FUNCTION_BLOCK TestAwaitChainNormal
VAR
	nState: UDINT := 0;
	await: Await;

	fbClient: FB_IotHttpClient := (
		sHostName:='localhost',
		bKeepAlive:=TRUE,
		tConnectionTimeout:=T#10S,
		nHostPort:=8000
	);
	
	fbRequest: FB_IotHttpRequest;
	sEndpoint: STRING := '/hello-world';
	response: STRING(255);

	fbJson: FB_JsonDomParser;
	
	jsonDoc: SJsonValue;
	jsonMember: SJsonValue;
	isJsonMemberString: BOOL;
	
	RisingEdge: R_TRIG;
	
	bSend: BOOL;
	requestSent: BOOL;
	cycleCounter: INT := 0;
	lenResponse: INT := 0;
	
	// Awaitable Errors
	onRequestError: OnRequestError := (errorName:='Request error', onErrorStep:=500);
	onResponseError: OnRequestError := (errorName:='Response error', onErrorStep:=500);
	onJsonError: OnJsonError := (errorName:='Json error', onErrorStep:=500);
	
	//Callbacks
	findJsonMemberCallback: FindJsonMember := 
	(
		jsonDomParser:=fbJson, 
		jsonReference:=jsonDoc,
		memberReference:=jsonMember
	);
	
	getJsonStringCallback: GetJsonString := 
	(
		jsonDomParser:=fbJson,
		bufferReference:=response,
		memberReference:=jsonMember
	);
	
	isJsonMemberStringCallback: IsJsonMemberString := 
	(
		jsonDomParser:=fbJson,
		memberReference:=jsonMember,
		isStringReference:=isJsonMemberString
	);
	
END_VAR

RisingEdge(CLK:= bSend );
fbClient.Execute();


CASE nState OF
	
	
	000: // Check if client is configured before moving on to the next step
		
		await.continueIf(fbClient.bConfigured);		
	
	
	010: // Waiting for input to start the request process
		
		await.continueIf(RisingEdge.Q);
	
	
	020: // Send the request
	
		cycleCounter := 0;
		
		requestSent := fbRequest.SendRequest(
			sUri:=sEndpoint, 
			fbClient:=fbClient, 
			eRequestType:=ETcIotHttpRequestType.HTTP_Get, 
			0, // payload, 
			0, // payload size  
			0  // header
		);
					
		await.catchIf(fbRequest.bError,onRequestError, 'An error occured while sending the request')
			.continueIf(requestSent);
	
	030: // Check if request was successful
	
		await.catchIf(fbRequest.bError,onRequestError, 'An error occured after sending the request')
			.continueIf(fbRequest.nStatusCode = 200);
			
		cycleCounter := cycleCounter + 1;
	
	040: // Get JsonDoc and on success call the findJsonMemberCallback

		jsonDoc := fbRequest.GetJsonDomContent(fbJson);
		findJsonMemberCallback.memberToFind := 'message';
		await.evalue(jsonDoc <> 0, findJsonMemberCallback, onJsonError, 'jsonDoc is an invalid pointer');

	050: //	Check if jsonMember is a valid pointer. On success call the isJsonMemberStringCallback
	
		await.evalue(jsonMember <> 0, isJsonMemberStringCallback, onJsonError, 'jsonMember is an invalid pointer');

		
	060: // Check the type of the json response value and on success call the getJsonStringCallback
		
		await.evalue(isJsonMemberString, getJsonStringCallback, onJsonError, 'The type of the message response is not String');
		
	070: // Check the len of the response
	
		await.evalue(len(response) > 0, 0, onResponseError, 'The length of the response is 0');
		
	500: // Error step

			
	
END_CASE

METHOD FB_init : BOOL
VAR_INPUT
	bInitRetains : BOOL; // if TRUE, the retain variables are initialized (warm start / cold start)
	bInCopyCode : BOOL;  // if TRUE, the instance afterwards gets moved into the copy code (online change)
END_VAR
await.setStepPointer := ADR(nState);
await.setIncreaseValue := 10;
END_METHOD

END_FUNCTION_BLOCK

(* stored: Version 1.1.0.1, ProductVersion 3.1.4024.12
   POU TestAwaitChainNormal: Id {a510cb06-81bf-437b-8803-498bf1e19fea}, SpecialFunc None
   Method FB_init: Id {602c78fd-7321-4821-a589-e6ae8f6a9170} *)
